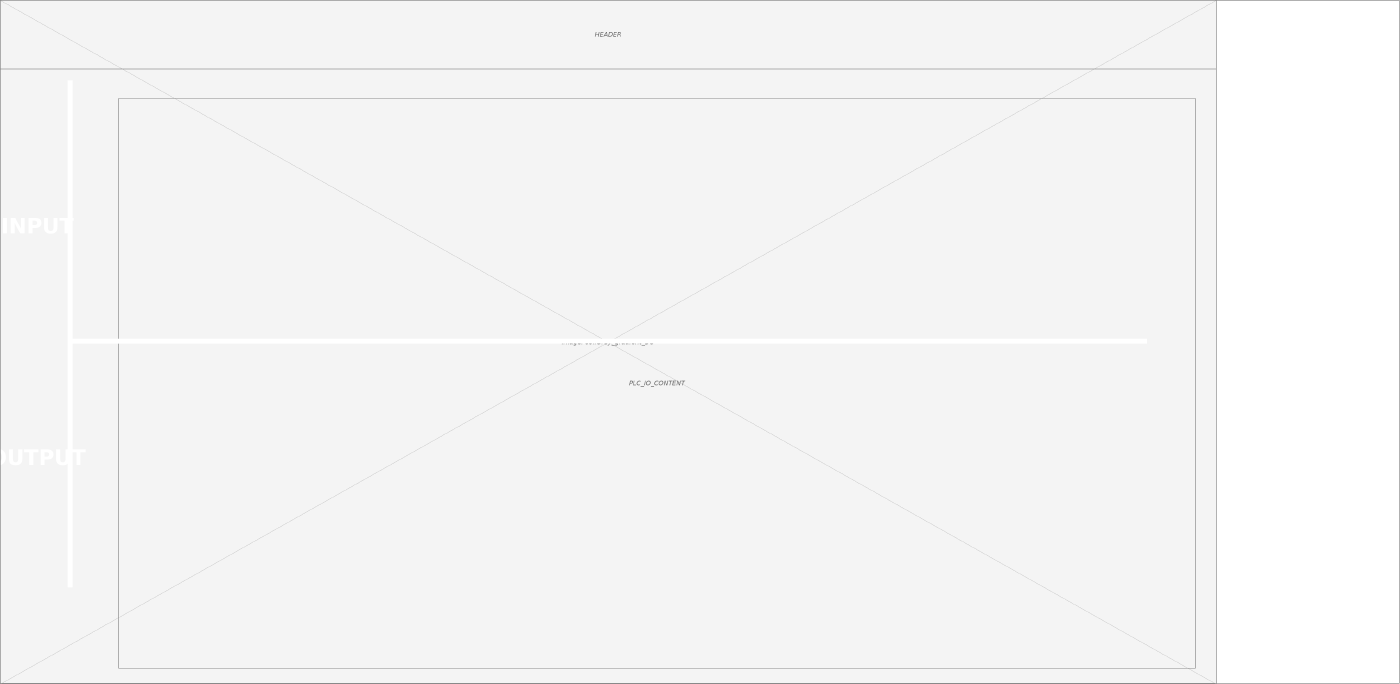
VISUALIZATION PLC_IO_PAGE  // 2210x1080
    Image (0,0 1920x1080), image: ImagePool.Grey_gradient_BG
    Frame (0,0 1920x109)
        shows HEADER()
    Rectangle (-55,320 229x74), angle 270, "INPUT"
    Rectangle (-290,524 800x7), angle 270
    Frame (187,155 1700x900)
        shows PLC_IO_CONTENT()
    Rectangle (110,535 1700x7)
    Rectangle (-70,685 258x74), angle 270, "OUTPUT"
END_VISUALIZATION

(* stored: Version 1.1.0.1, ProductVersion 3.1.4024.12
   Visu PLC_IO_PAGE: Id {ffdbce28-aca1-469c-8f44-6900024e00d2} *)
